// TIA Portal V17 export
// export: Created 2024-01-30T08:49:15.883956Z, ExportSetting WithDefaults, DisplayName Totally Integrated Automation Portal, DisplayVersion V17 Update 6, DisplayName TIA Portal Openness, DisplayVersion V17 Update 6, DisplayName TIA Portal Version Control Interface, DisplayVersion V17, DisplayName STEP 7 Professional, DisplayVersion V17 Update 6, DisplayName STEP 7 Safety, DisplayVersion V17 Update 6, DisplayName WinCC Advanced, DisplayVersion V17 Update 6
FUNCTION_BLOCK "Gatewas_RS232_LK_G5000"   // FB10, LAD
{ S7_Optimized_Access := 'TRUE' }
VERSION : 0.1
// stored: AutoNumber true, IsIECCheckEnabled false, IsRetainMemResEnabled false, MemoryReserve 100, SetENOAutomatically false, UDAEnableTagReadback false
   VAR_INPUT
      IN_COM : "UDT_LKG5000_RS232_RCV";
      IN_DATA : "UDT_RS232_RCV_DATA";
      SEND_TELEGRAM : Bool;
      COMMAND : String[10];
   END_VAR
   VAR_OUTPUT
      OUT_COM : "UDT_LKG5000_RS232_SEND";
      OUT_DATA : "UDT_RS232_SEND_DATA";
   END_VAR
   VAR
      COMMAND_SIGN : Array[0..10] of Char;
      Cnt_Command : UInt;
      IEC_Timer_0_Instance { S7_SetPoint := 'True'} : TOF_TIME;
      IEC_Timer_0_Instance_1 { S7_SetPoint := 'True'} : TOF_TIME;
   END_VAR
BEGIN

REGION Network 2 (SCL)
   Strg_TO_Chars(Strg:=#COMMAND,
                 pChars:=0,
                 Cnt=>#Cnt_Command,
                 Chars:=#COMMAND_SIGN);





   // Send frame
   #OUT_COM.Sendframe_size := 20;
   // Receive Frame
   #OUT_COM.Recvframe_size := 20;


   //#OUT_DATA.Data[0] := B#16#02;
   #OUT_DATA.Data[0] := #COMMAND_SIGN[0];
   #OUT_DATA.Data[1] := #COMMAND_SIGN[1];
   #OUT_DATA.Data[2] := #COMMAND_SIGN[2];
   #OUT_DATA.Data[3] := #COMMAND_SIGN[3];
   #OUT_DATA.Data[4] := #COMMAND_SIGN[4];
   #OUT_DATA.Data[5] :=  B#16#D0;

   //#OUT_DATA.Data[5] := #COMMAND_SIGN[5];
   //#OUT_DATA.Data[6] := #COMMAND_SIGN[6];
   //#OUT_DATA.Data[7] := #COMMAND_SIGN[7];
   //#OUT_DATA.Data[8] := #COMMAND_SIGN[8];
   //#OUT_DATA.Data[9] := #COMMAND_SIGN[9];
   //#OUT_DATA.Data[10] := #COMMAND_SIGN[10];
   //#OUT_DATA.Data[11] := #COMMAND_SIGN[11];
   //#OUT_DATA.Data[12] := #COMMAND_SIGN[12];
   //#OUT_DATA.Data[13] := #COMMAND_SIGN[13];
   //#OUT_DATA.Data[14] := #COMMAND_SIGN[14];
   //#OUT_DATA.Data[15] := #COMMAND_SIGN[15];
   //#OUT_DATA.Data[16] := #COMMAND_SIGN[16];
   //#OUT_DATA.Data[17] := #COMMAND_SIGN[17];
   //#OUT_DATA.Data[18] := #COMMAND_SIGN[18];
   //#OUT_DATA.Data[19] := #COMMAND_SIGN[19];
   //#OUT_DATA.Data[20] := #COMMAND_SIGN[20];
   //#OUT_DATA.Data[21] := #COMMAND_SIGN[21];
   //#OUT_DATA.Data[22] := #COMMAND_SIGN[22];
   //#OUT_DATA.Data[23] := B#16#D0;


   "R_TRIG_DB"(CLK:=#SEND_TELEGRAM);

   "IEC_Timer_0_DB".TP(IN:="R_TRIG_DB".Q,
                       PT:=T#2s);

   #OUT_COM.CTRL_Send := "IEC_Timer_0_DB".Q;


   "F_TRIG_DB"(CLK:=#OUT_COM.CTRL_Send);
END_REGION

REGION Network 3
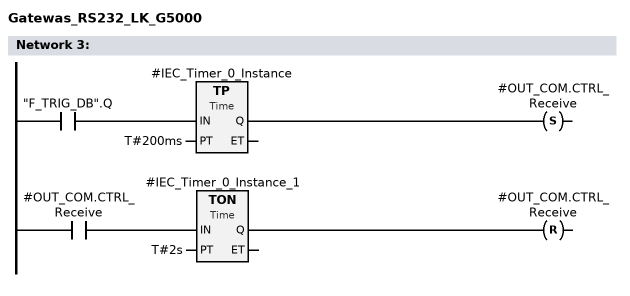
   RUNG wire#powerrail
      Contact( "F_TRIG_DB".Q )
      { S7_Templates := "time_type := Time" } #IEC_Timer_0_Instance.TP(pt := T#200ms, et =>)
      S_Coil( #OUT_COM.CTRL_Receive )
   END_RUNG
   RUNG wire#powerrail
      Contact( #OUT_COM.CTRL_Receive )
      { S7_Templates := "time_type := Time" } #IEC_Timer_0_Instance_1.TON(pt := T#2s, et =>)
      R_Coil( #OUT_COM.CTRL_Receive )
   END_RUNG
   // the same network as SCL:
   #IEC_Timer_0_Instance(IN := "F_TRIG_DB".Q, PT := T#200ms);   // TP
   IF #IEC_Timer_0_Instance.Q THEN #OUT_COM.CTRL_Receive := TRUE; END_IF;
   #IEC_Timer_0_Instance_1(IN := #OUT_COM.CTRL_Receive, PT := T#2s);   // TON
   IF #IEC_Timer_0_Instance_1.Q THEN #OUT_COM.CTRL_Receive := FALSE; END_IF;
END_REGION
END_FUNCTION_BLOCK
